// TwinCAT 3 PLC project txi_hxr_motion
// ProgramVersion: 3.1.4024.12
// libraries:
//   LCLS General, * (SLAC)
//   lcls-twincat-motion, * (SLAC)
//   lcls-twincat-physics, * (SLAC)
//   lcls2-cc-lib, * (SLAC)
//   PMPS, * (SLAC - LCLS)
//   Tc2_MC2, * (Beckhoff Automation GmbH)
//   Tc2_Standard, * (Beckhoff Automation GmbH)
//   Tc2_System, * (Beckhoff Automation GmbH)
//   Tc3_Module, * (Beckhoff Automation GmbH)
// project tree:
//   GVLs/ GVL.TcGVL (not stored), Main.TcGVL (not stored)
//   / PlcTask.TcTTO (not stored)
//   POUs/ PRG_AL1L1_L2SI.TcPOU (not stored), PRG_IM2L1_PPM.TcPOU, PRG_01_PLCTASK.TcPOU (not stored), PRG_SL3L1_SCATTER.TcPOU (not stored)
//   POUs/temp/ FB_SLITS.TcPOU (not stored), FB_SLITS_POWER.TcPOU (not stored), FB_SLITS_SCATTER.TcPOU (not stored)

// ---- POUs/PRG_IM2L1_PPM.TcPOU
PROGRAM PRG_IM2L1_PPM
VAR
        {attribute 'pytmc' := '
        pv: IM2L1:PPM
        io: io
    '}
    {attribute 'TcLinkTo' := '.fbGige.iIlluminatorINT := TIIB[IM2L1-EL4004]^AO Outputs Channel 1^Analog output;
                              .fbGige.bGigePower := TIIB[IM2L1-EL2004]^Channel 3^Output;
                              .fbPowerMeter.iVoltageINT := TIIB[IM2L1-EL3062]^AI Standard Channel 1^Value;
                              .fbPowerMeter.fbThermoCouple.bError := TIIB[IM2L1-EL3314]^TC Inputs Channel 1^Status^Error;
                              .fbPowerMeter.fbThermoCouple.bUnderrange := TIIB[IM2L1-EL3314]^TC Inputs Channel 1^Status^Underrange;
                              .fbPowerMeter.fbThermoCouple.bOverrange := TIIB[IM2L1-EL3314]^TC Inputs Channel 1^Status^Overrange;
                              .fbPowerMeter.fbThermoCouple.iRaw := TIIB[IM2L1-EL3314]^TC Inputs Channel 1^Value;
                              .fbYagThermoCouple.bError := TIIB[IM2L1-EL3314]^TC Inputs Channel 2^Status^Error;
                              .fbYagThermoCouple.bUnderrange := TIIB[IM2L1-EL3314]^TC Inputs Channel 2^Status^Underrange;
                              .fbYagThermoCouple.bOverrange := TIIB[IM2L1-EL3314]^TC Inputs Channel 2^Status^Overrange;
                              .fbYagThermoCouple.iRaw := TIIB[IM2L1-EL3314]^TC Inputs Channel 2^Value'}
    fbIM2L1: FB_PPM;

END_VAR

fbIM2L1.nTransitionAssertionID := 16#2110;
fbIM2L1.nUnknownAssertionID := 16#2119;

fbIM2L1.stOut.fPosition := -8.82;
fbIM2L1.stOut.bUseRawCounts := FALSE;
fbIM2L1.stOut.nRequestAssertionID := 16#2111;
fbIM2L1.stOut.stBeamParams := PMPS_GVL.cstFullBeam;
fbIM2L1.stOut.bValid := TRUE;

fbIM2L1.stPower.fPosition := -47.92;
fbIM2L1.stPower.bUseRawCounts := FALSE;
fbIM2L1.stPower.nRequestAssertionID := 16#2112;
fbIM2L1.stPower.stBeamParams := PMPS_GVL.cstFullBeam;
fbIM2L1.stPower.bValid := TRUE;

fbIM2L1.stYag1.fPosition := -71.92;
fbIM2L1.stYag1.bUseRawCounts := FALSE;
fbIM2L1.stYag1.nRequestAssertionID := 16#2113;
fbIM2L1.stYag1.stBeamParams := PMPS_GVL.cstFullBeam;
fbIM2L1.stYag1.bValid := TRUE;

fbIM2L1.stYag2.fPosition := -97.93;
fbIM2L1.stYag2.bUseRawCounts := FALSE;
fbIM2L1.stYag2.nRequestAssertionID := 16#2114;
fbIM2L1.stYag2.stBeamParams := PMPS_GVL.cstFullBeam;
fbIM2L1.stYag2.bValid := TRUE;

fbIM2L1(
    fbArbiter := GVL.fbArbiter1,
    fbFFHWO := GVL.fbFastFaultOutput1,
    stYStage := Main.M2);

END_PROGRAM
